// TIA Portal V16 export
// export: Created 2021-09-08T12:46:10.4767322Z, ExportSetting WithDefaults, DisplayName Totally Integrated Automation Portal, DisplayVersion V16 Update 3, DisplayName TIA Portal Version Control Interface, DisplayVersion V16 Update 2, DisplayName TIA Portal Openness, DisplayVersion V16 Update 3, DisplayName TIA Portal Teamcenter Gateway, DisplayVersion V16, DisplayName STEP 7 Professional, DisplayVersion V16 Update 3, DisplayName STEP 7 Safety, DisplayVersion V16, DisplayName WinCC Advanced, DisplayVersion V16 Update 3
DATA_BLOCK "AllAv_DB"   // DB3
VERSION : 0.1
// stored: AutoNumber true, DBAccessibleFromOPCUA true, InstanceOfName AllAv, InstanceOfType FB
"AllAv"
   // VAR
   //    DVM201 { S7_SetPoint := 'True'} : "AvCntrl";
   //    SOV801 { S7_SetPoint := 'True'} : "AvCntrl";
   //    SOV901 { S7_SetPoint := 'True'} : "AvCntrl";
   //    SOV902 { S7_SetPoint := 'True'} : "AvCntrl";
   //    SOV1301 { S7_SetPoint := 'True'} : "AvCntrl";
   //    SOV1302 { S7_SetPoint := 'True'} : "AvCntrl";
   //    SOV1303 { S7_SetPoint := 'True'} : "AvCntrl";
   //    DVA501 { S7_SetPoint := 'True'} : "AvCntrl";
   //    DVA502 { S7_SetPoint := 'True'} : "AvCntrl";
   //    DVA504 { S7_SetPoint := 'True'} : "AvCntrl";
   //    DVA505 { S7_SetPoint := 'True'} : "AvCntrl";
   //    DVA506 { S7_SetPoint := 'True'} : "AvCntrl";
   //    DVA507 { S7_SetPoint := 'True'} : "AvCntrl";
   //    DVA508 { S7_SetPoint := 'True'} : "AvCntrl";
   //    DVA509 { S7_SetPoint := 'True'} : "AvCntrl";
   //    DVA511 { S7_SetPoint := 'True'} : "AvCntrl";
   //    DVA512 { S7_SetPoint := 'True'} : "AvCntrl";
   //    DVA513 { S7_SetPoint := 'True'} : "AvCntrl";
   //    DVA514 { S7_SetPoint := 'True'} : "AvCntrl";
   //    DVA515 { S7_SetPoint := 'True'} : "AvCntrl";
   //    DVA516 { S7_SetPoint := 'True'} : "AvCntrl";
   //    DVA1801 { S7_SetPoint := 'True'} : "AvCntrl";
   // END_VAR
BEGIN
END_DATA_BLOCK
